TYPE Vec8di : ARRAY[1..8] OF DINT; END_TYPE

(* stored: Version 1.1.0.1, ProductVersion 3.1.4024.11
   DUT Vec8di: Id {2beac656-9a9c-4927-84b0-0b583bb1dd97} *)
